FUNCTION_BLOCK ML_model
  (* Version 1.0, 2005-09-20, Goran Cengic, Chalmers *)
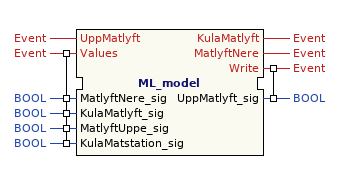
  EVENT_INPUT
    UppMatlyft;
    Values WITH MatlyftNere_sig, KulaMatlyft_sig, MatlyftUppe_sig, KulaMatstation_sig;
  END_EVENT
  EVENT_OUTPUT
    KulaMatlyft;
    MatlyftNere;
    Write WITH UppMatlyft_sig;
  END_EVENT
  VAR_INPUT
    MatlyftNere_sig : BOOL;
    KulaMatlyft_sig : BOOL;
    MatlyftUppe_sig : BOOL;
    KulaMatstation_sig : BOOL;
  END_VAR
  VAR_OUTPUT
    UppMatlyft_sig : BOOL;
  END_VAR
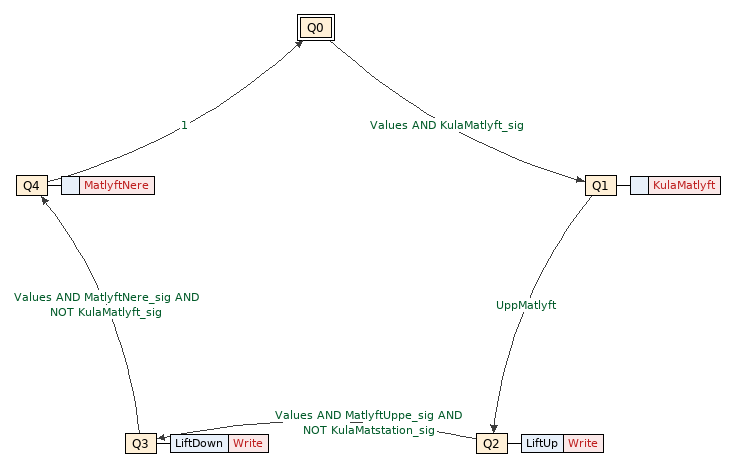
  EC_STATES
    Q0;
    Q1 : -> KulaMatlyft;
    Q2 : LiftUp -> Write;
    Q3 : LiftDown -> Write;
    Q4 : -> MatlyftNere;
  END_STATES
  EC_TRANSITIONS
    Q0 TO Q1 := Values AND KulaMatlyft_sig;
    Q1 TO Q2 := UppMatlyft;
    Q2 TO Q3 := Values AND MatlyftUppe_sig AND NOT KulaMatstation_sig;
    Q3 TO Q4 := Values AND MatlyftNere_sig AND NOT KulaMatlyft_sig;
    Q4 TO Q0 := 1;
  END_TRANSITIONS
  ALGORITHM LiftUp IN Java:
		System.out.println("Lifting ML up.");
		UppMatlyft_sig = true;
  END_ALGORITHM
  ALGORITHM LiftDown IN Java:
		System.out.println("Bringing ML down.");
		UppMatlyft_sig = false;
  END_ALGORITHM
END_FUNCTION_BLOCK
